FUNCTION_BLOCK WPsensorBA (* Composite Function Block Type *)
  (* Standard: 61499-2 *)
  (* Version 0.2, 2003-12-05, JHC, Rockwell Automation, Renamed from NEWCOMPFB. *)
  (* Version 0.1, 2002-01-08, JHC, Rockwell Automation, Added DLY FB as example. *)
  (* Version 0.0, 2000-05-27, JHC, Rockwell Automation *)
  (* Compiler header: package fb.rt.pnp; *)
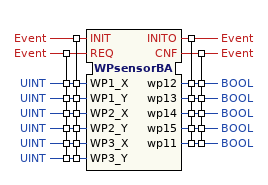
  EVENT_INPUT
    INIT WITH WP1_X, WP1_Y, WP2_X, WP2_Y, WP3_Y, WP3_X; (* Initialization Request *)
    REQ WITH WP1_Y, WP1_X, WP2_X, WP2_Y, WP3_X, WP3_Y; (* Normal Execution Request *)
  END_EVENT
  EVENT_OUTPUT
    INITO WITH wp12, wp14, wp11, wp13, wp15; (* Initialization Confirm *)
    CNF WITH wp12, wp13, wp14, wp11, wp15; (* Execution Confirmation *)
  END_EVENT
  VAR_INPUT
    WP1_X : UINT;
    WP1_Y : UINT;
    WP2_X : UINT;
    WP2_Y : UINT;
    WP3_X : UINT;
    WP3_Y : UINT;
  END_VAR
  VAR_OUTPUT
    wp12 : BOOL;
    wp13 : BOOL;
    wp14 : BOOL;
    wp15 : BOOL;
    wp11 : BOOL;
  END_VAR
  FBS
    WP1 : my_sensor2(zone1 := [529,539], zone2 := [383,393]);
    WP2 : my_sensor2(zone1 := [604,614], zone2 := [533,543]);
    WP3 : my_sensor2(zone1 := [679,689], zone2 := [458,468]);
    WP01 : my_sensor2(zone2 := [210,225], zone1 := [370,380]);
    WP02 : my_sensor2(zone2 := [210,225], zone1 := [370,380]);
    WP03 : my_sensor2(zone2 := [210,225], zone1 := [370,380]);
    WP0 : OR;
  END_FBS
  EVENT_CONNECTIONS
    INIT TO WP1.INIT;
    REQ TO WP1.REQ;
    REQ TO WP2.REQ;
    REQ TO WP3.REQ;
    WP1.INITO TO WP2.INIT;
    WP2.INITO TO WP3.INIT;
    WP1.CNF TO CNF;
    WP2.CNF TO CNF;
    WP3.CNF TO CNF;
    REQ TO WP01.REQ;
    WP01.INITO TO WP02.INIT;
    WP02.INITO TO WP03.INIT;
    REQ TO WP02.REQ;
    REQ TO WP03.REQ;
    WP03.CNF TO WP0.REQ;
    WP02.CNF TO WP0.REQ;
    WP01.CNF TO WP0.REQ;
    WP0.CNF TO CNF;
    WP3.INITO TO WP01.INIT;
    WP03.INITO TO WP0.INIT;
    WP0.INITO TO INITO;
  END_CONNECTIONS
  DATA_CONNECTIONS
    WP1.QO TO wp12;
    WP2.QO TO wp13;
    WP3.QO TO wp14;
    WP1_X TO WP1.In1;
    WP1_Y TO WP1.In2;
    WP2_X TO WP2.In1;
    WP2_Y TO WP2.In2;
    WP3_X TO WP3.In1;
    WP3_Y TO WP3.In2;
    WP1_X TO WP01.In1;
    WP1_Y TO WP01.In2;
    WP2_X TO WP02.In1;
    WP2_Y TO WP02.In2;
    WP3_X TO WP03.In1;
    WP3_Y TO WP03.In2;
    WP03.QO TO WP0.i3;
    WP02.QO TO WP0.i2;
    WP01.QO TO WP0.i1;
    WP0.o TO wp15;
  END_CONNECTIONS
END_FUNCTION_BLOCK
